FUNCTION_BLOCK FB_BeamParamFanout_1
VAR_INPUT
	{attribute 'TcLinkTo' := 'TIIB[PMPS_IF2]^IO Inputs^CurrentBP1'}
	i_stBP	AT %I* :	ST_BeamParamsReadback;
	{attribute 'TcLinkTo' := 'TIIB[PMPS_IF2]^SYNC Inputs^TxPDO toggle'}
	xTxPDO_toggle	AT 	%I* :	BIT;
	{attribute 'TcLinkTo' := 'TIIB[PMPS_IF2]^SYNC Inputs^TxPDO state'}
	xTxPDO_state	AT	%I*	:	BIT;
END_VAR
VAR_OUTPUT
	stBP	:	ST_BeamParamsReadback;
END_VAR
VAR
END_VAR

END_FUNCTION_BLOCK

(* stored: Version 1.1.0.1, ProductVersion 3.1.4022.12
   POU FB_BeamParamFanout_1: Id {80b3baef-43ba-0d0e-3ca3-03159f78ed90}, SpecialFunc None *)
